FUNCTION_BLOCK Valve_Analog
VAR_INPUT
	//Position Feedback from Valve
	Position_Feedback : REAL; 
	//Position Request from PLC Program
	Position_Request : REAL;
	//True when valve does not reach position in time
	Position_Fail : BOOL;
	//Where should the valve move when not on/in failure state
	Position_Faulted : REAL;
END_VAR
VAR_OUTPUT
	//Position Command to Device
	Position_Command : REAL;
END_VAR
VAR	
END_VAR
VAR // added by the converter: edge detectors and wires of the graphical bodies
    _w1, _w2 : BOOL;
END_VAR

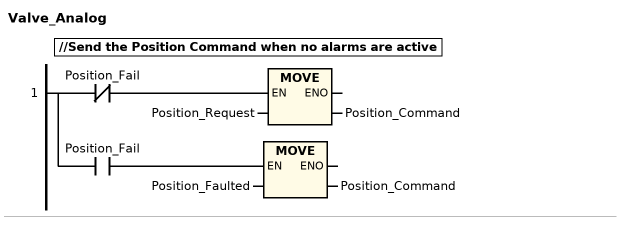
// NETWORK 1
// label: //Send the Position Command when no alarms are active
_w1 := NOT Position_Fail;
IF _w1 THEN Position_Command := Position_Request; END_IF
_w2 := Position_Fail;
IF _w2 THEN Position_Command := Position_Faulted; END_IF

END_FUNCTION_BLOCK

(* stored: Version 1.1.0.1, ProductVersion 3.1.4024.12
   POU Valve_Analog: Id {eb81a680-634a-469e-846c-a6f21734bdb6}, SpecialFunc None *)
